TYPE stBB02PL_Line EXTENDS stPIM_LineEventsModule :
STRUCT

	{attribute 'OPC.UA.DA' := '1'}
	stStation_BB02PL01 : stPIM_StationEventsModule_1_Machine;
END_STRUCT
END_TYPE

(* stored: Version 1.1.0.1, ProductVersion 3.1.4024.15
   DUT stBB02PL_Line: Id {2938061f-26cf-4efa-99a4-ea730bef982c} *)
